Staubli VAL3: Init.pgx

program Init()
begin

  clearBuffer(SocketUDP)
  resetMotion()

  launchAlter = true
  launchManualJoint = false
  launchToolChange = false

  OPCrxcmdOut = 0
  OPCrycmdOut = 0
  OPCrzcmdOut = 0
  FxLimit = 10
  FyLimit = 10
  FzLimit = 10
  OpcPrecisionMovement = 0.1
  OpcStepsRotation = 0.01
  OpcStepsMovement = 0.1
  OpcPreciseMode = false
  followHuman = false
  trAlterMove = {0,0,0,0,0,0}
  OPCGoHoming = false
  trAlter={0,0,0,0,0,0}
  delay(0)

end
